// TIA Portal V18 export
// export: Created 2025-12-01T12:38:52.3634353Z, ExportSetting None, DisplayName Totally Integrated Automation Portal, DisplayVersion V18 Update 5, DisplayName TIA Portal Openness, DisplayVersion V18 Update 5, DisplayName TIA Portal Teamcenter Gateway, DisplayVersion V18, DisplayName TIA Portal Version Control Interface, DisplayVersion V18, DisplayName STEP 7 Professional, DisplayVersion V18 Update 5, DisplayName STEP 7 Safety, DisplayVersion V18, DisplayName WinCC Professional, DisplayVersion V18 Update 5
DATA_BLOCK "Station4LoadData"   // DB516
{ S7_Optimized_Access := 'FALSE' }
// stored: AutoNumber false
   VAR
      "PLC.PartTypeID" : Int;
      "PLC.Station4RecipeNo" : Int;
      "PLC.Station4DMXCode" : String[128];
      "PLC.SubPartSN1" : String[128];
      "MES.ErrorCode" : Int;
      "MES.StatusBits" : DInt;
      "MES.Cycle_ID" : DInt;
      "MES.Unit_ParttypeID" : Int;
   END_VAR
BEGIN
END_DATA_BLOCK
